(* PLC project Unnamed, Unknown Unnamed 1 *)
(* stored: creationDateTime 2026-05-01T16:36:33, modificationDateTime 2026-05-01T18:09:33 *)

PROGRAM Project_01_Conveyor
  VAR
    PB_Start AT %IX0.0 : BOOL;
    PB_Stop AT %IX0.1 : BOOL;
    PB_EStop AT %IX0.2 : BOOL;
    PB_FaultReset AT %IX0.3 : BOOL;
    SW_ModeAuto AT %IX0.4 : BOOL;
    SEN_Entry AT %IX0.5 : BOOL;
    SEN_Exit AT %IX0.6 : BOOL;
    SEN_Jam AT %IX0.7 : BOOL;
    KM1_ConveyorMotor AT %QX0.0 : BOOL;
    HL1_RunLamp AT %QX0.1 : BOOL;
    HL2_AlarmLamp AT %QX0.2 : BOOL;
    HL3_AutoLamp AT %QX0.3 : BOOL;
    MR_RunLatch AT %M0.1 : BOOL;
    MR_FaultActive AT %M0.2 : BOOL;
    MR_AutoMode AT %M0.3 : BOOL;
    MR_ManualMode AT %M0.4 : BOOL;
    MR_AutoRunCmd AT %M0.5 : BOOL;
  END_VAR
  VAR
    MR_MasterEnable
     AT %M0.0 : BOOL;
  END_VAR
  VAR
    TON_JamDelay : TON;
    JamDelayTime : TIME := T#3s;
    AutoTimeoutTime : TIME := T#15s;
    TON_AutoTimeout : TON;
  END_VAR

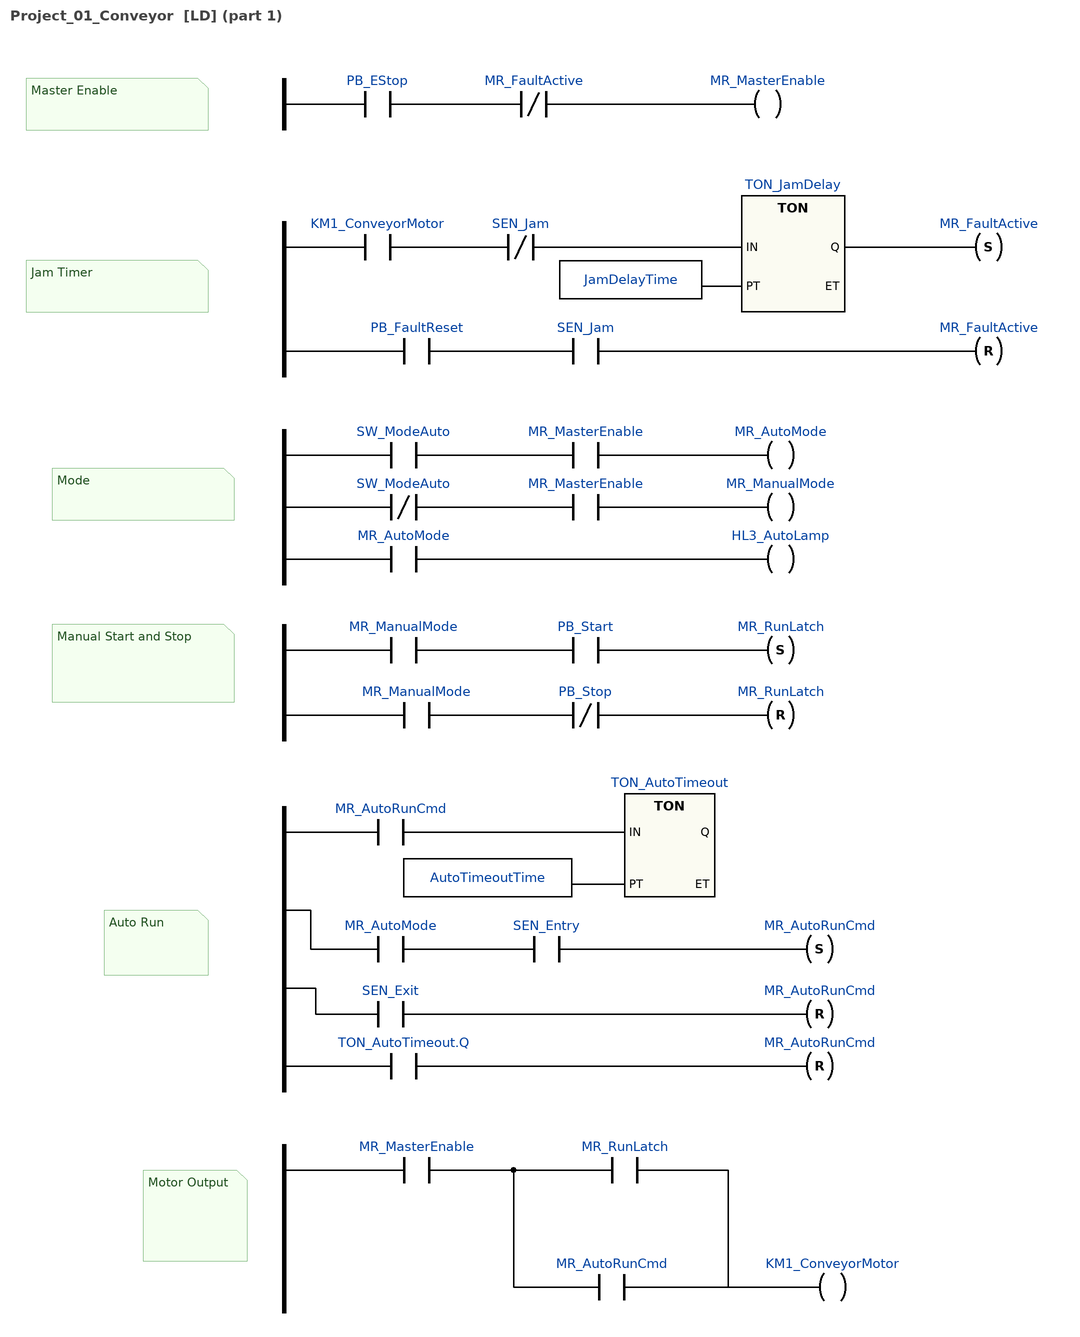
(* LD diagram, written out as Structured Text *)
(* Master Enable *)
MR_MasterEnable := PB_EStop AND NOT MR_FaultActive;
TON_JamDelay(IN := KM1_ConveyorMotor AND NOT SEN_Jam, PT := JamDelayTime);
IF TON_JamDelay.Q THEN MR_FaultActive := TRUE; END_IF;
(* Jam Timer *)
IF PB_FaultReset AND SEN_Jam THEN MR_FaultActive := FALSE; END_IF;
MR_AutoMode := SW_ModeAuto AND MR_MasterEnable;
(* Mode *)
MR_ManualMode := NOT SW_ModeAuto AND MR_MasterEnable;
HL3_AutoLamp := MR_AutoMode;
(* Manual Start and Stop *)
IF MR_ManualMode AND PB_Start THEN MR_RunLatch := TRUE; END_IF;
IF MR_ManualMode AND NOT PB_Stop THEN MR_RunLatch := FALSE; END_IF;
(* Auto Run *)
IF MR_AutoMode AND SEN_Entry THEN MR_AutoRunCmd := TRUE; END_IF;
IF SEN_Exit THEN MR_AutoRunCmd := FALSE; END_IF;
IF TON_AutoTimeout.Q THEN MR_AutoRunCmd := FALSE; END_IF;
(* Motor Output *)
KM1_ConveyorMotor := MR_MasterEnable AND (MR_AutoRunCmd OR MR_RunLatch);
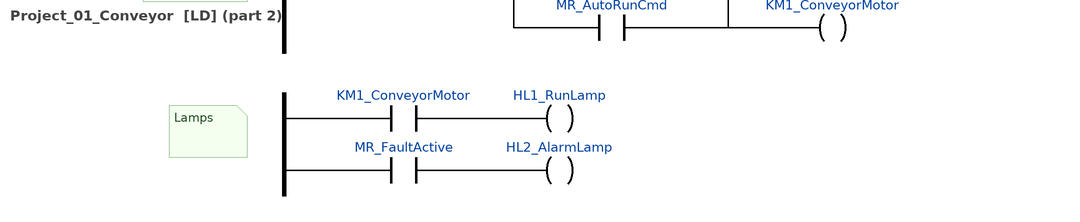
(* Lamps *)
HL1_RunLamp := KM1_ConveyorMotor;
HL2_AlarmLamp := MR_FaultActive;
TON_AutoTimeout(IN := MR_AutoRunCmd, PT := AutoTimeoutTime);
END_PROGRAM

CONFIGURATION Config0
  RESOURCE Res0 ON PLC
    TASK task0(INTERVAL := T#20ms, PRIORITY := 0);
    PROGRAM instance0 WITH task0 : Project_01_Conveyor;
  END_RESOURCE
END_CONFIGURATION
